PROGRAM MAIN
VAR
	iCounter : INT;
	bToggle		: BOOL;
	bReset		: BOOL;
	sText		: STRING;
	
	stMyType		: ST_MyType;
	
END_VAR


IF bToggle THEN
	sText := 'stop';
	iCounter := (iCounter + 1) MOD 1000;
	IF iCounter = 0 THEN
		bToggle := FALSE;
	END_IF
ELSE
	sText := 'start';
	IF bReset THEN
		bReset := FALSE;
		iCounter := 0;
	END_IF	
END_IF

Alarming();
AlarmingEx();
AlarmExtension();

END_PROGRAM

(* stored: Version 1.1.0.1, ProductVersion 3.1.4024.12
   POU MAIN: Id {ff167503-42de-46b6-a4f4-dbe0042569ea}, SpecialFunc None *)
